INTERFACE iContainTraceArgument EXTENDS iBase

{attribute 'monitoring' := 'call'}
PROPERTY Arguments : iTraceArgument
GET
END_GET
END_PROPERTY

END_INTERFACE

(* stored: Version 1.1.0.1, ProductVersion 3.1.4026.18
   Itf iContainTraceArgument: Id {1e6cdb11-1e0e-0439-0cb0-9fbc821de5d0}
   Property Arguments: Id {b2c6d343-6151-0f57-1d9e-02097bc270d1}
   Get Get: Id {837180dc-4ddb-0457-1c2a-d13856d5b2f1} *)
